{attribute 'qualified_only'}
{attribute 'strict'}
{attribute 'to_string'}
TYPE ENUM_InternalControl_StateMachine :
(
	READY := 0, 
	STANDBY,
	RUN,
	FAULT
);
END_TYPE

(* stored: Version 1.1.0.1
   DUT ENUM_InternalControl_StateMachine: Id {d787d589-610b-4e31-8201-1fc09ee3908e} *)
